(* IEC 61131-3 sources: Industry-PLC-LLM/data/PLCBEAD_repo/PLCBEAD_PLCEmbed-main/PLC-BEAD/Source/GEB/MIX, 1 file *)

(* ---- MIX.ST ---- *)
FUNCTION MIX:REAL

	VAR_INPUT
		A :	REAL;
		B :	REAL;
		M :	REAL;
	END_VAR

	MIX := (1.0 - M) * A + M * B;

END_FUNCTION

PROGRAM program0
	VAR
		A :	REAL;
		B :	REAL;
		M :	REAL;

		OUT : REAL;
	END_VAR

	OUT := MIX(A, B, M);

END_PROGRAM
